(* PLC project Generated.project, CODESYS CODESYS V3.5 SP19 Patch 1 *)
(* stored: creationDateTime 2026-09-06T13:00:42.571904, modificationDateTime 2026-09-06T13:00:42.571904 *)

TYPE ST_PreflightHMI : STRUCT
  BtnRun : BOOL;
  PreflightOk : BOOL;
  PreflightDone : BOOL;
  PreflightBusy : BOOL;
  PreflightErrorId : WORD;
END_STRUCT;
END_TYPE
